FUNCTION FC_LimitMaxReal : bool
VAR_INPUT
	iMaster:		REAL;
END_VAR
VAR_IN_OUT
	ioSlave:		REAL;
END_VAR

IF (ioSlave > iMaster) THEN
	ioSlave := iMaster;
END_IF

END_FUNCTION

(* stored: Version 1.1.0.1, ProductVersion 3.1.4026.18
   POU FC_LimitMaxReal: Id {3e0e7137-2360-4404-8715-11fd187bde79}, SpecialFunc None *)
